PROGRAM P3_07_SendReport
VAR
	fbSend				:FB_PythonScript;
	
	iError				:INT;
	tonResetError		:TON;
	
	iStep				:INT;
END_VAR

VAR PERSISTENT
	
END_VAR

tonResetError(IN:=(iError<>0),PT:=T#3S);
IF tonResetError.Q THEN
	iError:=0;
END_IF
CASE iStep OF
	
	0:
		IF GV.stReport.bStartSend_Sequence THEN
			GV.stReport.bStartSend_Sequence:=FALSE;
			iError:=0;
			iStep:=10;
		END_IF
	
	10:
		GV.stReport.bSend_Report:=TRUE;
		IF fbSend.q_bBusy THEN
			iStep:=15;
		END_IF
	
	15:
		IF NOT fbSend.q_bBusy AND fbSend.q_bDone THEN
			iStep:=999;
		ELSIF fbSend.q_bError THEN
			iError:=iStep;
			iStep:=999;
		END_IF
	
	999:
		iStep:=0;
END_CASE
ACT_CMDs();

ACTION ACT_CMDs:
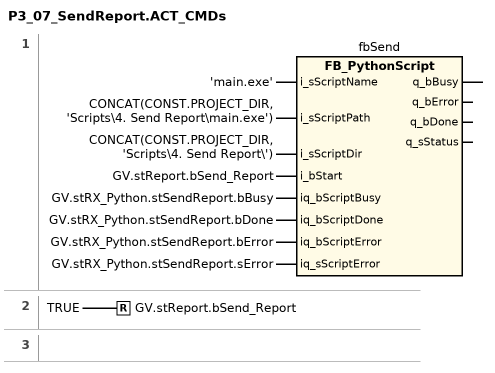
// NETWORK 1
fbSend(
    i_sScriptName := 'main.exe',
    i_sScriptPath := CONCAT(CONST.PROJECT_DIR,'Scripts\4. Send Report\main.exe'),
    i_sScriptDir := CONCAT(CONST.PROJECT_DIR,'Scripts\4. Send Report\'),
    i_bStart := GV.stReport.bSend_Report,
    iq_bScriptBusy := GV.stRX_Python.stSendReport.bBusy,
    iq_bScriptDone := GV.stRX_Python.stSendReport.bDone,
    iq_bScriptError := GV.stRX_Python.stSendReport.bError,
    iq_sScriptError := GV.stRX_Python.stSendReport.sError); // FB_PythonScript

// NETWORK 2
GV.stReport.bSend_Report R= TRUE;

// NETWORK 3
END_ACTION

END_PROGRAM

(* stored: Version 1.1.0.1, ProductVersion 3.1.4024.12
   POU P3_07_SendReport: Id {c2f9588a-ef92-420f-a595-be8635af2707}, SpecialFunc None
   Action ACT_CMDs: Id {e9907169-23b2-4aa5-a35a-35258428c632} *)
